{attribute 'qualified_only'}
VAR_GLOBAL
		EtherCAT_Master_ATxxxx : EtherCAT_Master_ATxxxx_981D2C79;
END_VAR

(* stored: Version 1.2.0.0, ProductVersion 3.1.4024.11
   GVL GVL_iXlinker: Id {c94a0b48-ec8c-434e-b01e-da93ba87e0ce} *)
